TYPE ST_WarehouseGetBox :
STRUCT
	//倉儲儲位
	StorageInfor	:INT;
	//盒子順序
	BoxOrder 		:INT;
END_STRUCT
END_TYPE

(* stored: Version 1.1.0.1, ProductVersion 3.1.4024.13
   DUT ST_WarehouseGetBox: Id {2cb6daff-fe16-4cf0-bdb8-146a90208e88} *)
